Universal Robots PolyScope program: Return_kettle.urp

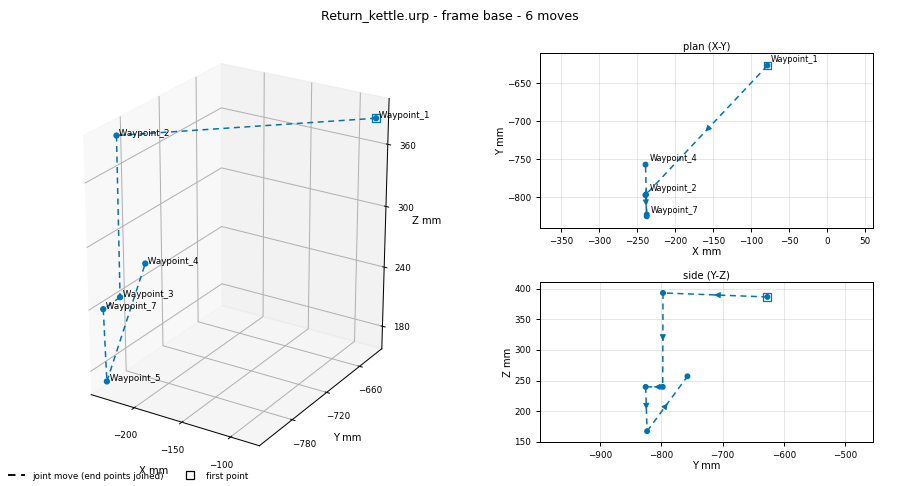
[picture p0: tool path of Return_kettle.urp in frame base, 6 of 6 moves have a stored position in this frame; points joined in program order, loops and branches not executed]
Program Return_kettle (installation=default directory=/programs/Matcha createdIn=5.12.6.1102099 lastSavedIn=5.12.6.1102099 robotSerialNumber=20215500597)
Calibrated DH parameters: a=[0.000193, -0.066673, -0.391568, -0.000012, 0.00005, 0]; d=[0.162643, -472.05677, 465.132521, 7.058239, 0.099746, 0.099582]; alpha=[1.571116, 0.00089, 0.003862, 1.569269, -1.569248, 0]; deltaTheta=[0, -1.413394, 7.628392, 0.068187, 0, -0.000001]
Robot Program (runOnlyOnce=true)
  MoveJ speed 60 deg/s, acceleration 80 deg/s^2 (useActiveTCP=true) feature=Base
    Waypoint Waypoint_1: TCP in base x=-78.557 y=-626.96 z=386.248 mm, rx=0.0116 ry=-2.2035 rz=2.2302 rad; joints [53.981, -98.506, 113.327, -15.857, 53.985, 180.128] deg; TCP offset x=0 y=0 z=191.5 mm, rx=0 ry=0 rz=0 rad
    Waypoint Waypoint_2: TCP in base x=-238.787 y=-797.019 z=392.782 mm, rx=0.0285 ry=-2.2147 rz=2.2269 rad; joints [50.629, -68.308, 78.056, -10.361, 49.922, 179.708] deg
    Waypoint Waypoint_3: TCP in base x=-238.838 y=-797.498 z=239.747 mm, rx=0.0286 ry=-2.2147 rz=2.2269 rad; joints [50.65, -61.161, 91.273, -30.71, 50.011, 179.683] deg
    Waypoint Waypoint_7: TCP in base x=-237.351 y=-825.318 z=239.668 mm, rx=-0.0012 ry=2.1548 rz=-2.2647 rad; joints [52.593, -57.948, 88.245, -34.097, 52.079, 182.991] deg
    Waypoint Waypoint_5: TCP in base x=-237.34 y=-822.9 z=167.475 mm, rx=-0.0013 ry=2.1549 rz=-2.2647 rad; joints [52.443, -52.647, 91.804, -42.951, 51.953, 182.979] deg
    URCap Gripper (Robotiq_Grippers, Robotiq Inc.) dataModel(position=49.80392156862745, force=100.0, speed=64.0, positionInDouble=49.80392156862745, forceInDouble=100.0, speedInDouble=64.0, slaveIds=[9], blocking=true)
    Waypoint Waypoint_4: TCP in base x=-238.915 y=-757.22 z=256.922 mm, rx=0.0287 ry=-2.2144 rz=2.227 rad; joints [47.776, -66.671, 96.927, -30.893, 47.141, 179.719] deg
    SafeHome (positionOptionType=SPEED_AND_ACCELERATION speed=1.047198 acceleration=1.396263 nextMotionTime=2)
